{attribute 'GeneratedUsingTerminal: EM3701-0000-0016'}
{attribute addProperty BoxType "EM3701-0000-0016"}
{attribute addProperty Id "EtcSlaveTerminalBaseAI_InputsAT %I*AI_Inputs_5AF6604E8WcStateAT %I*WcState_9091E0EB2InfoDataAT %I*InfoData_32EB74EA10"}
{attribute addProperty CRC "177471275"}
{attribute addProperty Size "20"}
TYPE EM3701_0A93FF2B EXTENDS EtcSlaveTerminalBase :
STRUCT
	{attribute addProperty Name "AI_Inputs"}
	AI_Inputs : AI_Inputs_5AF6604E;
	{attribute addProperty Name "WcState"}
	WcState : WcState_9091E0EB;
	{attribute addProperty Name "InfoData"}
	InfoData : InfoData_32EB74EA;
END_STRUCT
END_TYPE

(* stored: Version 1.2.0.0, ProductVersion 3.1.4024.9
   DUT EM3701_0A93FF2B: Id {620ae656-5e75-47f4-923d-437dc597afb1} *)
